Yaskawa INFORM job: WELDING-BACK-ST-2.JBI

/JOB
//NAME WELDING-BACK-ST-2
//POS
///NPOS 0,0,0,0,0,0
//INST
///DATE 2018/11/22 17:18
///ATTR SC,RW
NOP
IFTHEN D005=8
	'***** CMF100
	 CALL JOB:WELDING-CMF100-ST2-BACK
ENDIF
IFTHEN D005=4
	'***** F........ sensors
	 CALL JOB:WELDING-F-SENSORS-BACK-ST2
ENDIF
END
